// TIA Portal V19 export
VAR_GLOBAL   // PLC tag table "00_A03_MB3_Tower"
   A03_TowerHorn_SL301 AT %Q302.1 : Bool;   // 372HA1
   A03_TowerLampYellow_SL301 AT %Q301.7 : Bool;   // 372HL1
   A03_TowerLampWhite_SL301 AT %Q302.0 : Bool;   // 372HL2
   A03_Segnalazione_Scarico_Pezzi_Accoppiati_Blu_SL302 AT %Q302.2 : Bool;   // 373HL1
   A03_Segnalazione_Scarico_Pacco__Blu_SL303 AT %Q351.7 : Bool;   // 374HL1
   A03_Segnalazione_Stato_Barriera_Interna_Bianco_SL304 AT %Q352.0 : Bool;   // 374HL2
   MB3_Pb_Reset_Anomalie AT %I113.0 : Bool;   // 310SH1
   MB3_Pb_Manuale_Area03 AT %I113.1 : Bool;   // 310SA1
   MB3_Pb_Automatico_Area03 AT %I113.2 : Bool;   // 310SA1
   MB3_Pb_Start_Ciclo_Area03 AT %I113.3 : Bool;   // 310SH2
   MB3_Pb_Stop_Ciclo_Area03 AT %I113.4 : Bool;   // 310SB1
   MB3_Pb_Start_Ciclo_Area02 AT %I113.5 : Bool;   // 310SH3
   MB3_Pb_Stop_Ciclo_Area02 AT %I113.6 : Bool;   // 310SB2
   MB3_Pb_Start_Ciclo_Area01 AT %I113.7 : Bool;   // 311SH1
   MB3_Pb_Stop_Ciclo_Area01 AT %I114.0 : Bool;   // 311SB1
   MB3_Pb_Avanti_Stazione_3_Area03 AT %I114.1 : Bool;   // 311SH2
   MB3_Pb_Avanti_Stazione_4_Area03 AT %I114.2 : Bool;   // 311SH3
   MB3_Pb_Avanti_Stazione_2_Area03 AT %I114.3 : Bool;   // 311SH4
   MB3_Pb_Avanti_Stazione_1_Area03 AT %I114.4 : Bool;   // 311SH5
   MB3_Pb_Comando_Manuale_Jog_Plus_A03 AT %I114.5 : Bool;   // 311SA1
   MB3_Pb_Comando_Manuale_Jog_Minus_A03 AT %I114.6 : Bool;   // 311SA1
   MB3_Pb_Avanti_Pezzo_Area02 AT %I114.7 : Bool;   // 312SB1
   MB3_Lp_Reset_Anomalie AT %Q111.6 : Bool;   // 310SH1
   MB3_Lp_Abilitazione_Automatico_Area03 AT %Q111.7 : Bool;   // 310HL1
   MB3_Lp_Start_Ciclo_Area03 AT %Q112.0 : Bool;   // 310SH2
   MB3_Lp_Start_Ciclo_Area02 AT %Q112.1 : Bool;   // 310SH3
   MB3_Lp_Start_Ciclo_Area01 AT %Q112.2 : Bool;   // 311SH1
   MB3_Lp_Avanti_Stazione_3_Area03 AT %Q112.3 : Bool;   // 311SH2
   MB3_Lp_Avanti_Stazione_4_Area03 AT %Q112.4 : Bool;   // 311SH3
   MB3_Lp_Avanti_Stazione_2_Area03 AT %Q112.5 : Bool;   // 311SH4
   MB3_Lp_Avanti_Stazione_1_Area03 AT %Q112.6 : Bool;   // 311SH5
   MB3_Lp_Comando_Manuale_Jog_Plus AT %Q112.7 : Bool;   // 311SA1
   MB3_Lp_LIBERO AT %Q122.5 : Bool;   // 312 - LIBERO
   MB3_Pb_Comando_Manuale_Jog_Plus_A04 AT %I143.0 : Bool;   // 311SA1
   MB3_Pb_Comando_Manuale_Jog_Minus_A04 AT %I143.1 : Bool;   // 311SA1
   MB3_Pb_Start_Ciclo_Area04 AT %I142.5 : Bool;   // 312SH1
   MB3_Pb_Stop_Ciclo_Area04 AT %I142.6 : Bool;   // 312SB2
   MB3_Pb_Manuale_Area04 AT %I115.0 : Bool;   // 312SA1
   MB3_Pb_Automatico_Area04 AT %I115.1 : Bool;   // 312SA1
   MB3_Lp_Abilitazione_Automatico_Area04 AT %Q113.0 : Bool;   // 312HL1
   MB3_Lp_Comando_Manuale_Jog_Plus_A04 AT %Q122.6 : Bool;   // 312SA2
   A04_TowerHorn_SL401 AT %Q303.6 : Bool;   // 372HA1
   A04_TowerLampYellow_SL401 AT %Q303.4 : Bool;   // 372HL1
   A04_TowerLampWhite_SL401 AT %Q303.5 : Bool;   // 372HL2
END_VAR
